FUNCTION_BLOCK FB_Cylinder EXTENDS TcoCore.TcoComponent IMPLEMENTS I_Cyl_Move, I_Cyl_Diag, I_Cyl_AtHome, I_Cyl_AtWork
VAR_INPUT
	In : ST_Cyl_inputs;
END_VAR
VAR_OUTPUT
	Out : ST_Cyl_inputs;
END_VAR
VAR
	Config:	ST_Cyl_Config;
	Control: ST_Cyl_Control;
	Status: ST_Cyl_Status;
	Diag: ST_Cyl_Diagnosis;
END_VAR

M_Diag();

METHOD M_Diag : E_Diag
VAR_INPUT
END_VAR
// NETWORK 1
END_METHOD

METHOD M_MoveToHome : BOOL
VAR_INPUT
END_VAR
END_METHOD

METHOD M_MoveToWork : BOOL
VAR_INPUT
END_VAR
END_METHOD

PROPERTY P_AtHome : BOOL
GET
END_GET
END_PROPERTY

PROPERTY P_AtWork : BOOL
GET
END_GET
END_PROPERTY

END_FUNCTION_BLOCK

(* stored: Version 1.1.0.1, ProductVersion 3.1.4024.6
   POU FB_Cylinder: Id {40aaf20f-d296-0a95-19c9-968f23726cd4}, SpecialFunc None
   Method M_Diag: Id {31845e9a-5247-0060-112f-cef81fdfb14c}
   Method M_MoveToHome: Id {d9de80c4-0891-0ff4-125b-274a305bea46}
   Method M_MoveToWork: Id {7d8d7a6b-6b02-044e-3184-d5c39196a959}
   Property P_AtHome: Id {936aeeba-1842-0581-3d16-7c46cd3001a5}
   Get Get: Id {57043cd7-3c2d-0fff-2991-8c87d77f94c9}
   Property P_AtWork: Id {281a410a-a660-0540-228a-e5b631a1cc6d}
   Get Get: Id {96f4ce80-2b64-09ae-2cc0-06fab131ac21} *)
